Omron CX-Programmer project NewProject (CX-Programmer 9.70)

# PLC NewPLC1: CJ1M CPU11

## Program NewProgram1 (cyclic task 0)
Local symbols
ETAPA_0 W0.00 BOOL  ; Inicio
ETAPA_1 W0.01 BOOL  ; Ligar motor
ETAPA_2 W0.02 BOOL  ; Desligar motor
FLAG_TEMP T0000 BOOL  ; Temporizador
KM1 100.00 BOOL  ; Contactor
START 0.00 BOOL  ; START
STOP 0.01 BOOL  ; STOP
TEMPO #100 NUMBER  ; Tempo temporizador 10 segundos
TEMPORIZADOR_2 1 NUMBER  ; Temporizador 2

### Section START

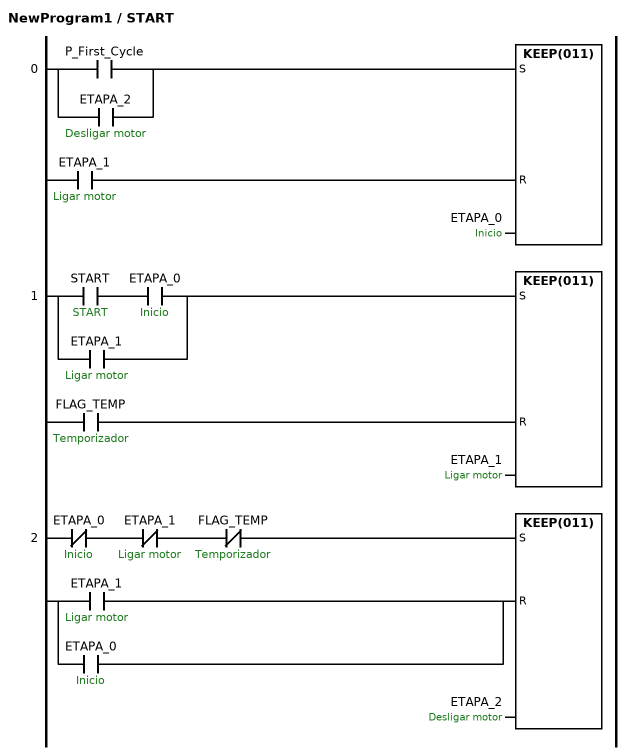
; rung 0
LD P_First_Cycle
OR ETAPA_2  ; Desligar motor
LD ETAPA_1  ; Ligar motor
KEEP(011) ETAPA_0  ; Inicio
; rung 1
LD START  ; START
AND ETAPA_0  ; Inicio
OR ETAPA_1  ; Ligar motor
LD FLAG_TEMP  ; Temporizador
KEEP(011) ETAPA_1  ; Ligar motor
; rung 2
LDNOT ETAPA_0  ; Inicio
ANDNOT ETAPA_1  ; Ligar motor
ANDNOT FLAG_TEMP  ; Temporizador
LD ETAPA_1  ; Ligar motor
OR ETAPA_0  ; Inicio
KEEP(011) ETAPA_2  ; Desligar motor

### Section END
; rung 0
END(001)